PROGRAM POU
VAR
END_VAR

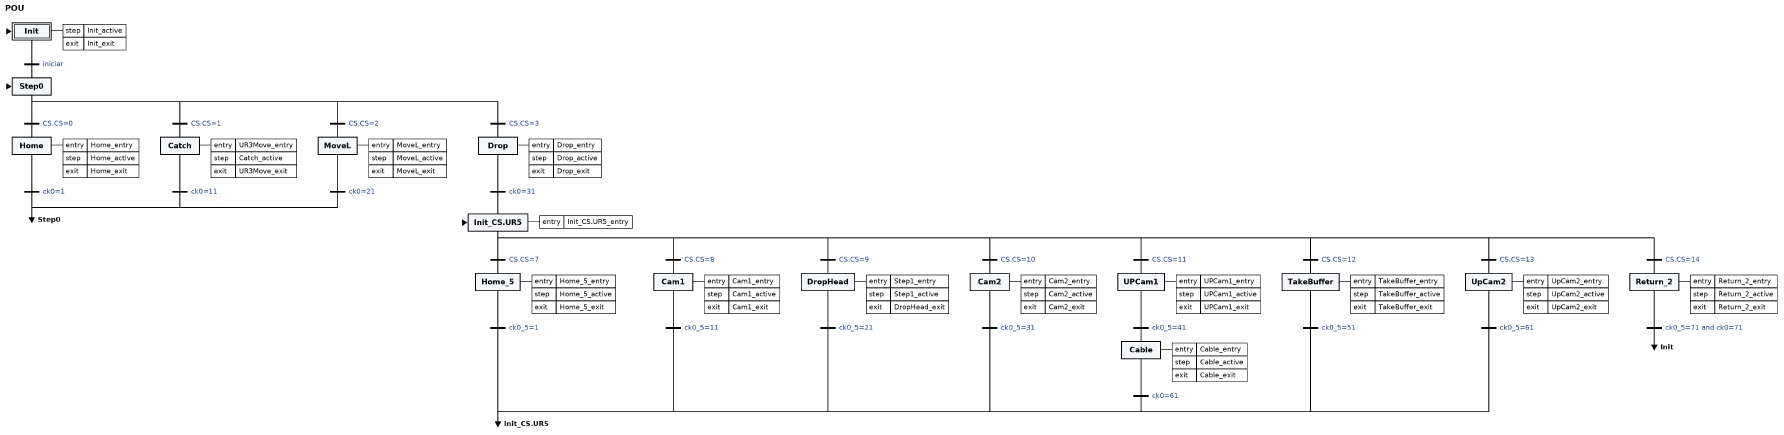
INITIAL_STEP Init:
    Init_active(N);  // step action
    Init_exit(P0);  // exit action
END_STEP
TRANSITION FROM Init TO Step0
    := iniciar;
END_TRANSITION
STEP Step0:
END_STEP
TRANSITION FROM Step0 TO Home
    := CS.CS=0;
END_TRANSITION
STEP Home:
    Home_entry(P1);  // entry action
    Home_active(N);  // step action
    Home_exit(P0);  // exit action
END_STEP
TRANSITION FROM Home TO Step0
    := ck0=1;
END_TRANSITION
TRANSITION FROM Step0 TO Catch
    := CS.CS=1;
END_TRANSITION
STEP Catch:
    UR3Move_entry(P1);  // entry action
    Catch_active(N);  // step action
    UR3Move_exit(P0);  // exit action
END_STEP
TRANSITION FROM Catch TO Step0
    := ck0=11;
END_TRANSITION
TRANSITION FROM Step0 TO MoveL
    := CS.CS=2;
END_TRANSITION
STEP MoveL:
    MoveL_entry(P1);  // entry action
    MoveL_active(N);  // step action
    MoveL_exit(P0);  // exit action
END_STEP
TRANSITION FROM MoveL TO Step0
    := ck0=21;
END_TRANSITION
TRANSITION FROM Step0 TO Drop
    := CS.CS=3;
END_TRANSITION
STEP Drop:
    Drop_entry(P1);  // entry action
    Drop_active(N);  // step action
    Drop_exit(P0);  // exit action
END_STEP
TRANSITION FROM Drop TO Init_CS_UR5
    := ck0=31;
END_TRANSITION
STEP Init_CS_UR5:  // name as stored: Init_CS.UR5
    Init_CS.UR5_entry(P1);  // entry action
END_STEP
TRANSITION FROM Init_CS_UR5 TO Home_5
    := CS.CS=7;
END_TRANSITION
STEP Home_5:
    Home_5_entry(P1);  // entry action
    Home_5_active(N);  // step action
    Home_5_exit(P0);  // exit action
END_STEP
TRANSITION FROM Home_5 TO Init_CS_UR5
    := ck0_5=1;
END_TRANSITION
TRANSITION FROM Init_CS_UR5 TO Cam1
    := CS.CS=8;
END_TRANSITION
STEP Cam1:
    Cam1_entry(P1);  // entry action
    Cam1_active(N);  // step action
    Cam1_exit(P0);  // exit action
END_STEP
TRANSITION FROM Cam1 TO Init_CS_UR5
    := ck0_5=11;
END_TRANSITION
TRANSITION FROM Init_CS_UR5 TO DropHead
    := CS.CS=9;
END_TRANSITION
STEP DropHead:
    Step1_entry(P1);  // entry action
    Step1_active(N);  // step action
    DropHead_exit(P0);  // exit action
END_STEP
TRANSITION FROM DropHead TO Init_CS_UR5
    := ck0_5=21;
END_TRANSITION
TRANSITION FROM Init_CS_UR5 TO Cam2
    := CS.CS=10;
END_TRANSITION
STEP Cam2:
    Cam2_entry(P1);  // entry action
    Cam2_active(N);  // step action
    Cam2_exit(P0);  // exit action
END_STEP
TRANSITION FROM Cam2 TO Init_CS_UR5
    := ck0_5=31;
END_TRANSITION
TRANSITION FROM Init_CS_UR5 TO UPCam1
    := CS.CS=11;
END_TRANSITION
STEP UPCam1:
    UPCam1_entry(P1);  // entry action
    UPCam1_active(N);  // step action
    UPCam1_exit(P0);  // exit action
END_STEP
TRANSITION FROM UPCam1 TO Cable
    := ck0_5=41;
END_TRANSITION
STEP Cable:
    Cable_entry(P1);  // entry action
    Cable_active(N);  // step action
    Cable_exit(P0);  // exit action
END_STEP
TRANSITION FROM Cable TO Init_CS_UR5
    := ck0=61;
END_TRANSITION
TRANSITION FROM Init_CS_UR5 TO TakeBuffer
    := CS.CS=12;
END_TRANSITION
STEP TakeBuffer:
    TakeBuffer_entry(P1);  // entry action
    TakeBuffer_active(N);  // step action
    TakeBuffer_exit(P0);  // exit action
END_STEP
TRANSITION FROM TakeBuffer TO Init_CS_UR5
    := ck0_5=51;
END_TRANSITION
TRANSITION FROM Init_CS_UR5 TO UpCam2
    := CS.CS=13;
END_TRANSITION
STEP UpCam2:
    UpCam2_entry(P1);  // entry action
    UpCam2_active(N);  // step action
    UpCam2_exit(P0);  // exit action
END_STEP
TRANSITION FROM UpCam2 TO Init_CS_UR5
    := ck0_5=61;
END_TRANSITION
TRANSITION FROM Init_CS_UR5 TO Return_2
    := CS.CS=14;
END_TRANSITION
STEP Return_2:
    Return_2_entry(P1);  // entry action
    Return_2_active(N);  // step action
    Return_2_exit(P0);  // exit action
END_STEP
TRANSITION FROM Return_2 TO Init
    := ck0_5=71 and ck0=71;
END_TRANSITION

END_PROGRAM

(* stored: Version 1.1.0.1, ProductVersion 3.1.4024.4
   POU POU: Id {9ffd7d0d-d16b-4ef5-860d-dd1fc015e9aa}, SpecialFunc None *)
